INTERFACE I_PersistentEventStorage

METHOD StoreEvent
VAR_INPUT
	stEvent : ST_Event;
END_VAR
END_METHOD

END_INTERFACE

(* stored: Version 1.1.0.1, ProductVersion 3.1.4024.12
   Itf I_PersistentEventStorage: Id {b7720615-8b65-4262-a66f-4cdf59a365ce}
   Method StoreEvent: Id {714618a5-2ec1-4534-b328-3d942c0454a1} *)
